Universal Robots URScript: 4-movep.script

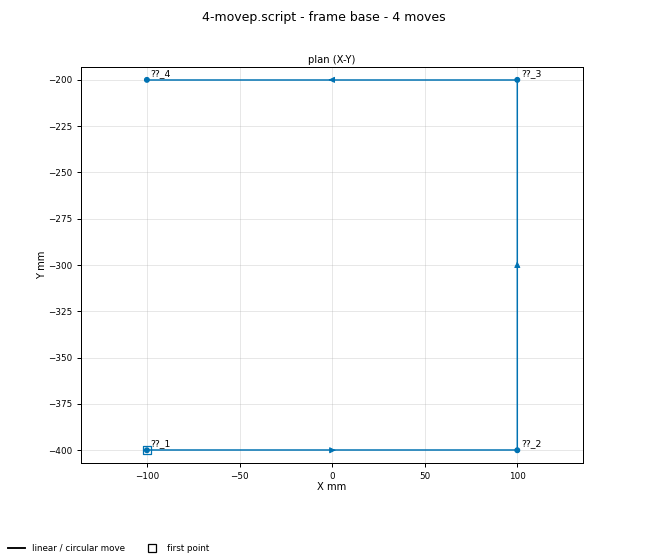
[picture p0: tool path of 4-movep.script in frame base, 4 of 4 moves have a stored position in this frame; points joined in program order, loops and branches not executed]
def P4movep():
  set_standard_analog_input_domain(0, 1)
  set_standard_analog_input_domain(1, 1)
  set_tool_analog_input_domain(0, 1)
  set_tool_analog_input_domain(1, 1)
  set_analog_outputdomain(0, 0)
  set_analog_outputdomain(1, 0)
  set_tool_voltage(0)
  set_tcp(p[0.0,0.0,0.0,0.0,0.0,0.0])
  set_payload(0.0)
  set_gravity([0.0, 0.0, 9.82])
  while (True):
    $ 1 "机器人程序"
    $ 2 "MoveP"
    $ 3 "路点_1"
    movep(p[-.100000000660, -.400000001042, .199999998231, -.001220983028, 3.116276481241, .038891916168], a=1.2, v=0.25, r=0.025)
    $ 4 "路点_2"
    movep(p[.099999906565, -.400000029719, .199999839972, -.001220578145, 3.116276713993, .038892761160], a=1.2, v=0.25, r=0.025)
    $ 5 "路点_3"
    movep(p[.100000030930, -.199999977208, .200000020249, -.001220905867, 3.116276536037, .038892034429], a=1.2, v=0.25, r=0.025)
    $ 6 "路点_4"
    movep(p[-.100000000341, -.199999999659, .199999839636, -.001221229174, 3.116276825727, .038892683103], a=1.2, v=0.25, r=0.025)
  end
end
